# EPICS StreamDevice protocol: stanford_sr400_photon_counterSup/stanford_sr400_photon_counter.proto
Terminator = CR LF;

getStatusByte {
    out "SS";
    in "%u";
}

getCounterA {
    out "QA";
    in "%d";
}

getCounterB {
    out "QB";
    in "%d";
}

startCounting {
    out "CS";
}

stopCounting {
    out "CH";
}

resetCounters {
    out "CR";
}
